FUNCTION_BLOCK ANYToJSON (* Transform 61499 types to JSON format *)
  (* Standard: 61499-2; Description: Copyright (c) 2018 fortiss GmbH This program and the accompanying materials are made available under the terms of the Eclipse Public License 2.0 which is available at https://www.eclipse.org/legal/epl-2.0/ SPDX-License-Identifier: EPL-2.0 *)
  (* Version 1.0, 2018-09-21, Jose Cabral, fortiss GmbH *)
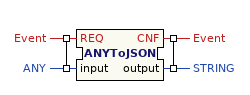
  EVENT_INPUT
    REQ WITH input; (* Request transformation *)
  END_EVENT
  EVENT_OUTPUT
    CNF WITH output; (* Transformation finished *)
  END_EVENT
  VAR_INPUT
    input : ANY; (* Input to be transformed *)
  END_VAR
  VAR_OUTPUT
    output : STRING; (* JSON transformation from input *)
  END_VAR
  (* Service APPLICATION/RESOURCE: Transform 61499 types to JSON format *)
END_FUNCTION_BLOCK
